FUNCTION_BLOCK TrainHA
  (* Standard: 61499-2 *)
  (* Version 0.1, 2017-00-29, hpea485, UOA *)
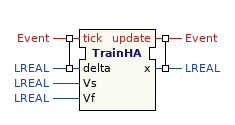
  EVENT_INPUT
    tick WITH delta;
  END_EVENT
  EVENT_OUTPUT
    update WITH x;
  END_EVENT
  VAR_INPUT
    delta : LREAL;
    Vs : LREAL;
    Vf : LREAL;
  END_VAR
  VAR_OUTPUT
    x : LREAL;
  END_VAR
  VAR
    Variable1 : BOOL;
  END_VAR
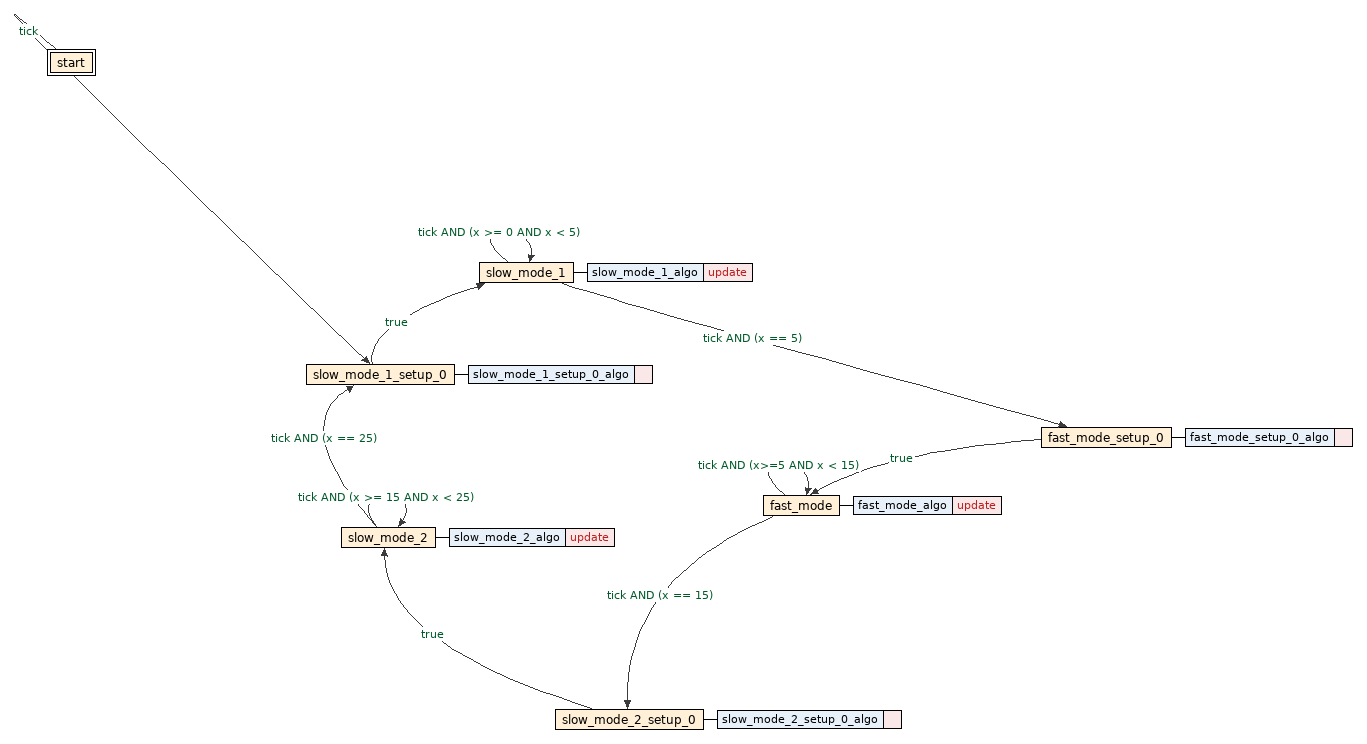
  EC_STATES
    start;
    slow_mode_1_setup_0 : slow_mode_1_setup_0_algo; (* ODE_init *)
    slow_mode_1 : slow_mode_1_algo -> update; (* x >= 0 AND x <= 5 *)
    fast_mode : fast_mode_algo -> update; (* x >= 5 AND x <= 15 *)
    slow_mode_2 : slow_mode_2_algo -> update; (* x >= 15 AND x <= 25 *)
    fast_mode_setup_0 : fast_mode_setup_0_algo; (* ODE_init *)
    slow_mode_2_setup_0 : slow_mode_2_setup_0_algo; (* ODE_init *)
  END_STATES
  EC_TRANSITIONS
    start TO slow_mode_1_setup_0 := tick;
    slow_mode_1 TO slow_mode_1 := tick AND (x >= 0 AND x < 5);
    slow_mode_1 TO fast_mode_setup_0 := tick AND (x == 5);
    fast_mode TO fast_mode := tick AND (x>=5 AND x < 15);
    fast_mode TO slow_mode_2_setup_0 := tick AND (x == 15);
    slow_mode_2 TO slow_mode_2 := tick AND (x >= 15 AND x < 25);
    slow_mode_2 TO slow_mode_1_setup_0 := tick AND (x == 25);
    fast_mode_setup_0 TO fast_mode := true;
    slow_mode_2_setup_0 TO slow_mode_2 := true;
    slow_mode_1_setup_0 TO slow_mode_1 := true;
  END_TRANSITIONS
  ALGORITHM fast_mode_algo IN C: (* ODE *)
x_dot = Vf;
  END_ALGORITHM
  ALGORITHM slow_mode_1_algo IN C: (* ODE *)
x_dot = Vs;
  END_ALGORITHM
  ALGORITHM slow_mode_2_algo IN C: (* ODE *)
x_dot = Vs;
  END_ALGORITHM
  ALGORITHM fast_mode_setup_0_algo IN C: (* ODE_init *)
ode = fast_mode_algo;
x_prime = x;
x_zero = x;
  END_ALGORITHM
  ALGORITHM slow_mode_2_setup_0_algo IN C: (* ODE_init *)
ode = slow_mode_2_algo;
x_prime = x;
x_zero = x;
  END_ALGORITHM
  ALGORITHM slow_mode_1_setup_0_algo IN C: (* ODE_init *)
ode = slow_mode_1_algo;
x_prime = 0;
x_zero = x;
  END_ALGORITHM
END_FUNCTION_BLOCK
